INTERFACE itfCommand

METHOD Abort : MC_Error
END_METHOD

PROPERTY Active : BOOL
GET
END_GET
END_PROPERTY

PROPERTY Busy : BOOL
GET
END_GET
END_PROPERTY

PROPERTY Command : MC_COMMAND_REF
GET
END_GET
END_PROPERTY

PROPERTY CommandAborted : BOOL
GET
END_GET
END_PROPERTY

PROPERTY Done : BOOL
GET
END_GET
END_PROPERTY

PROPERTY Error : BOOL
GET
END_GET
END_PROPERTY

PROPERTY ErrorId : MC_Error
GET
END_GET
END_PROPERTY

METHOD Wait : MC_Error
VAR_INPUT
	Timeout: TIME;
	AbortOnTimeout: BOOL;
END_VAR
END_METHOD

END_INTERFACE

(* stored: Version 1.1.0.1, ProductVersion 3.1.4024.12
   Itf itfCommand: Id {808308aa-5be1-474f-9cd7-f693a8f9904a}
   Method Abort: Id {8b5e35ac-b5b0-4aa3-ac23-dd574710cbdb}
   Property Active: Id {ee573e9a-5ea0-49eb-8a77-58c3db89cb06}
   Get Get: Id {c4c0014a-9026-4b8a-9650-13184f5bdc66}
   Property Busy: Id {219c6516-004b-45fc-b650-7ed67eb9c5f4}
   Get Get: Id {fd4f74cd-a0ae-4ec7-bbfa-8a862e2c0a66}
   Property Command: Id {75a96964-1bda-4b50-a0bc-30c1d7adea11}
   Get Get: Id {43c0171f-d1ec-4b63-a8af-eeaa97140843}
   Property CommandAborted: Id {1228aed1-e6c8-4a0c-83a8-614a39b5cd17}
   Get Get: Id {ceecb89e-362a-4f0a-a73b-7ba6f4a6410c}
   Property Done: Id {d40ac11d-8d91-4f20-b524-e82b3a89ff64}
   Get Get: Id {d8022f53-a405-4ef5-9214-73662c938099}
   Property Error: Id {3c0e0fa2-bc73-41b1-b093-306901cd5baf}
   Get Get: Id {42ae53d1-41e8-4672-9e91-39c95fd67e67}
   Property ErrorId: Id {fef3784f-c132-4b1e-9f11-d65718464c45}
   Get Get: Id {33e69af0-83b7-4144-822d-6b756181da67}
   Method Wait: Id {14133628-3c21-4d21-a48c-496a1b395288} *)
